FUNCTION_BLOCK FB_Axis
VAR_INPUT
	enable : BOOL;
	disable : BOOL;
	reset : BOOL;
END_VAR
VAR_OUTPUT
	iState : I_State := fbIdleState;
END_VAR
VAR
	fbIdleState : FB_Idle(THIS);
	fbErrorState : FB_Error(THIS);
	fbEnabledState : FB_Enabled(THIS);
	
	
END_VAR

IF enable THEN
	THIS^.iState.Enable();
END_IF
IF disable THEN
	THIS^.iState.Disable();
END_IF
IF reset THEN
	THIS^.iState.Reset();
END_IF

PROPERTY INTERNAL EnabledState : i_state
GET
EnabledState := THIS^.fbEnabledState;
END_GET
END_PROPERTY

PROPERTY INTERNAL ErrorState : i_state
GET
ErrorState := THIS^.fbErrorState;
END_GET
END_PROPERTY

PROPERTY INTERNAL IdleState : i_state
GET
IdleState := THIS^.fbIdleState;
END_GET
END_PROPERTY

METHOD INTERNAL SetState : BOOL
VAR_INPUT
	newState : I_State;
END_VAR
THIS^.iState := newState;
END_METHOD

END_FUNCTION_BLOCK

(* stored: Version 1.1.0.1, ProductVersion 3.1.4024.3
   POU FB_Axis: Id {c140482e-603b-4d92-ba54-92c858058e3b}, SpecialFunc None
   Property EnabledState: Id {5ffeb8a1-fdb6-49ee-8a62-4b69ce850e8e}
   Get Get: Id {07a91ee3-fb83-4c6b-86ef-5029fddacbc7}
   Property ErrorState: Id {b6d64575-3120-46eb-a886-6bc5f4a30c7c}
   Get Get: Id {920cef53-3a7f-4dfb-8999-78c716311f1a}
   Property IdleState: Id {5f667966-a52b-4199-ae09-c32b538fafa3}
   Get Get: Id {b9a52243-2ed4-470d-9f45-fec0b88b4391}
   Method SetState: Id {39e18b0d-168d-472d-8855-270e35112728} *)
